FUNCTION_BLOCK Monitoring_Error
VAR_INPUT
	negDirB	:	BOOL;
	posDirB	:	BOOL;
	command	:	REAL;
END_VAR
VAR_OUTPUT
	currentError	:	BOOL;
END_VAR

enableSolenoidControl(enaNegDir := negDirB, enaPosDir := posDirB, error := currentError);
commandCheck(comm := command, error := currentError);

METHOD PRIVATE commandCheck
VAR_INPUT
	comm : REAL;
END_VAR
VAR_IN_OUT
	error: BOOL;
END_VAR

IF ((comm <= 1000) AND (comm >0)) THEN
		IF posDirB THEN
			error := FALSE;
			generalVariable.staus.bError[2].showError := FALSE;
			ELSE
				error := TRUE;
				showError(2,'příkaz a směr se neshodují');
				END_IF;
	ELSIF ((comm >= -1000) AND (comm < 0)) THEN
			IF negDirB THEN
				error := FALSE;
				generalVariable.staus.bError[2].showError := FALSE;
			ELSE
				error := TRUE;
				showError(2,'příkaz a směr se neshodují');
				END_IF;
			ELSIF comm = 0 THEN
				generalVariable.staus.Standstill := TRUE;
				IF NOT(negDirB AND posDirB) THEN
					error := FALSE;
					generalVariable.staus.bError[3].showError := FALSE;
				ELSE
					error := TRUE;
					showError(3,'zahrnoval některé směry');       
				END_IF;
			END_IF;
END_METHOD

METHOD PRIVATE enableSolenoidControl
VAR_INPUT
	enaPosDir : BOOL;
	enaNegDir : BOOL;	
END_VAR
VAR_IN_OUT
	error: BOOL;
END_VAR
VAR
	strr	:	STRING;
END_VAR

IF (enaNegDir AND enaPosDir) THEN
	// error 
	currentError := TRUE;
	showError(1,'muze být aktivní pouze jedna cívka (PosDir nebo NegDir)');
	//errCode(1);
	ELSE
		currentError := FALSE ;
		generalVariable.staus.bError[1].showError := FALSE;
		END_IF
END_METHOD

METHOD PRIVATE showError
VAR_INPUT
	id	:	INT;
	str	:	STRING;
END_VAR
generalVariable.staus.bError[50].showError := FALSE;
IF NOT(generalVariable.staus.bError[id].showError) THEN
	generalVariable.staus.nErrorId[id] := id;
	generalVariable.staus.bError[id].errorName := str;
	generalVariable.staus.bError[id].showError := TRUE;
	blockMessage(str);
	END_IF;
END_METHOD

END_FUNCTION_BLOCK

(* stored: Version 1.1.0.1, ProductVersion 3.1.4024.12
   POU Monitoring_Error: Id {ddbe3727-6a6b-4e90-b0ef-5962f195c134}, SpecialFunc None
   Method commandCheck: Id {e37482b3-3f45-49ac-9845-c74e88b1bb1e}
   Method enableSolenoidControl: Id {612b163a-2352-495f-9f4e-55f73d756558}
   Method showError: Id {3873f583-cd35-46ae-a32e-68d649424b0b} *)
